PROGRAM MAIN
VAR
	Lesson_2_2 : FN_2_2_Finite_State_Machine;
END_VAR

Lesson_2_2();

END_PROGRAM

(* stored: Version 1.1.0.1, ProductVersion 3.1.4024.13
   POU MAIN: Id {0d3e2942-f68d-453c-b4a1-c0350d874497}, SpecialFunc None *)
